// TIA Portal V17 export
// export: Created 2025-07-01T09:58:31.5693186Z, ExportSetting WithDefaults, DisplayName Totally Integrated Automation Portal, DisplayVersion V17 Update 8, DisplayName TIA Portal Openness, DisplayVersion V17 Update 8, DisplayName TIA Portal Version Control Interface, DisplayVersion V17, DisplayName SINAMICS Startdrive Advanced, DisplayVersion V17 SP2, DisplayName SINAMICS Startdrive G110M, G120, G120C, G120D, G120P, G115D, DisplayVersion V17 SP2, DisplayName SINAMICS Startdrive G130, G150, S120, S150, SINAMICS MV, S210, DisplayVersion V17 SP2, DisplayName STEP 7 Professional, DisplayVersion V17 Update 8, DisplayName SINUMERIK ONE STEP 7 Toolbox, DisplayVersion V17 Update 12, DisplayName SINUMERIK ONE PLC Basic Program Plus, DisplayVersion V17 Update 12, DisplayName SINUMERIK 840D sl STEP 7 Toolbox, DisplayVersion V17 Update 12, DisplayName STEP 7 Safety, DisplayVersion V17 Update 6, DisplayName WinCC Advanced, DisplayVersion V17 Update 8
FUNCTION "FC15500_BDE" : Void   // FC15500, LAD
{ S7_Optimized_Access := 'TRUE' }
VERSION : 0.1
// stored: AutoNumber false, IsIECCheckEnabled false, SetENOAutomatically false, UDAEnableTagReadback false
BEGIN

REGION Network 1: FEED PART STATUS
   // PART_A/PART_B/PART_C/PART_D/PART_E
   // If the bit for the status of a feed part is to 0, the corresponding message text+ is available
   // is displayed in the image.
   // If the bit for the status of a feed part is set to 1, the corresponding message text + not available is displayed on the screen.
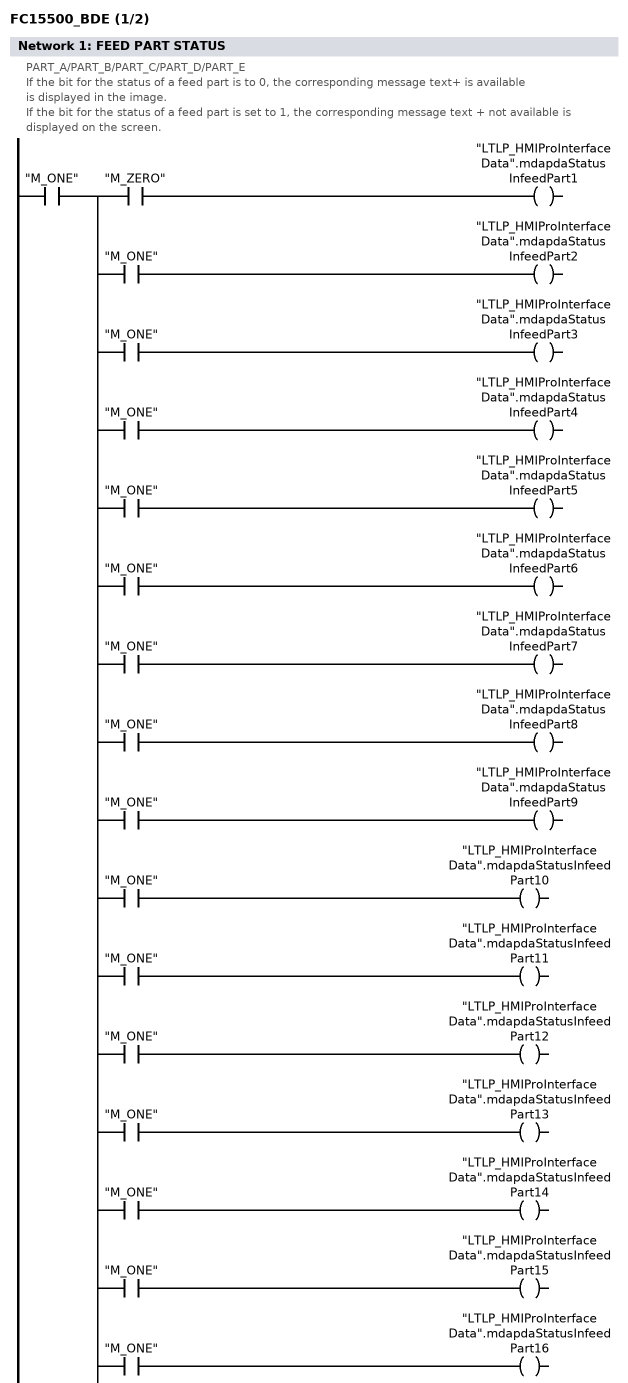
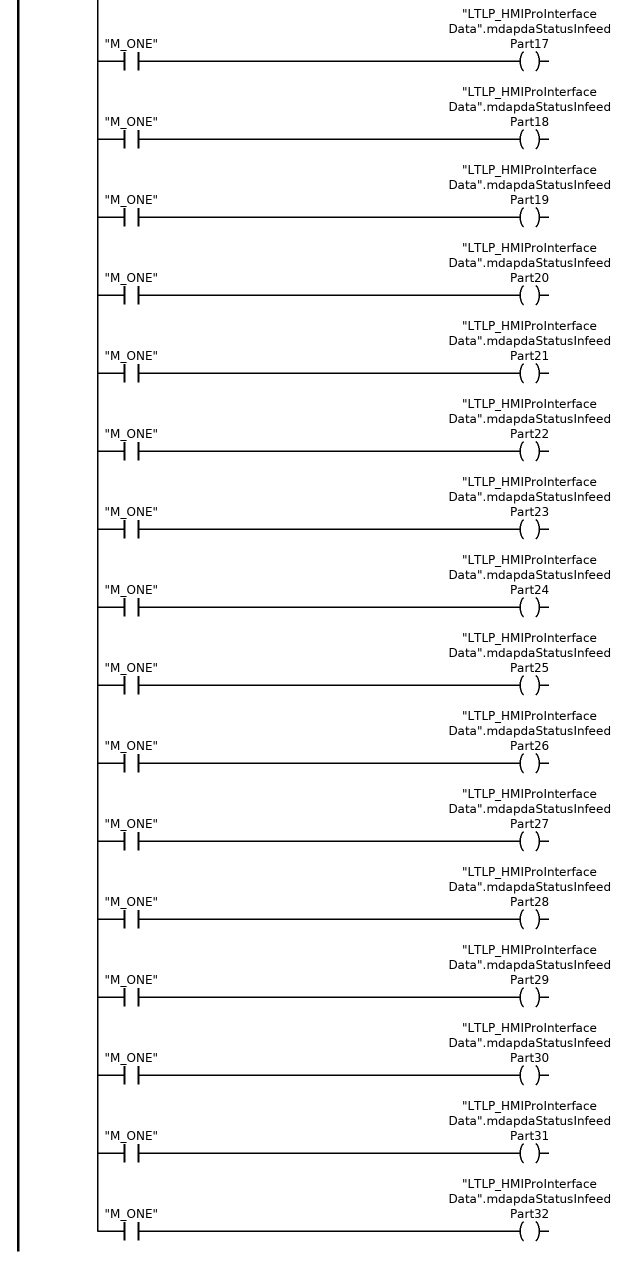
   RUNG wire#powerrail
      Contact( "M_ONE" )
      wire#w1
      Contact( "M_ZERO" )
      Coil( "LTLP_HMIProInterfaceData".mdapdaStatusInfeedPart1 )
   END_RUNG
   RUNG wire#w1
      Contact( "M_ONE" )
      Coil( "LTLP_HMIProInterfaceData".mdapdaStatusInfeedPart2 )
   END_RUNG
   RUNG wire#w1
      Contact( "M_ONE" )
      Coil( "LTLP_HMIProInterfaceData".mdapdaStatusInfeedPart3 )
   END_RUNG
   RUNG wire#w1
      Contact( "M_ONE" )
      Coil( "LTLP_HMIProInterfaceData".mdapdaStatusInfeedPart4 )
   END_RUNG
   RUNG wire#w1
      Contact( "M_ONE" )
      Coil( "LTLP_HMIProInterfaceData".mdapdaStatusInfeedPart5 )
   END_RUNG
   RUNG wire#w1
      Contact( "M_ONE" )
      Coil( "LTLP_HMIProInterfaceData".mdapdaStatusInfeedPart6 )
   END_RUNG
   RUNG wire#w1
      Contact( "M_ONE" )
      Coil( "LTLP_HMIProInterfaceData".mdapdaStatusInfeedPart7 )
   END_RUNG
   RUNG wire#w1
      Contact( "M_ONE" )
      Coil( "LTLP_HMIProInterfaceData".mdapdaStatusInfeedPart8 )
   END_RUNG
   RUNG wire#w1
      Contact( "M_ONE" )
      Coil( "LTLP_HMIProInterfaceData".mdapdaStatusInfeedPart9 )
   END_RUNG
   RUNG wire#w1
      Contact( "M_ONE" )
      Coil( "LTLP_HMIProInterfaceData".mdapdaStatusInfeedPart10 )
   END_RUNG
   RUNG wire#w1
      Contact( "M_ONE" )
      Coil( "LTLP_HMIProInterfaceData".mdapdaStatusInfeedPart11 )
   END_RUNG
   RUNG wire#w1
      Contact( "M_ONE" )
      Coil( "LTLP_HMIProInterfaceData".mdapdaStatusInfeedPart12 )
   END_RUNG
   RUNG wire#w1
      Contact( "M_ONE" )
      Coil( "LTLP_HMIProInterfaceData".mdapdaStatusInfeedPart13 )
   END_RUNG
   RUNG wire#w1
      Contact( "M_ONE" )
      Coil( "LTLP_HMIProInterfaceData".mdapdaStatusInfeedPart14 )
   END_RUNG
   RUNG wire#w1
      Contact( "M_ONE" )
      Coil( "LTLP_HMIProInterfaceData".mdapdaStatusInfeedPart15 )
   END_RUNG
   RUNG wire#w1
      Contact( "M_ONE" )
      Coil( "LTLP_HMIProInterfaceData".mdapdaStatusInfeedPart16 )
   END_RUNG
   RUNG wire#w1
      Contact( "M_ONE" )
      Coil( "LTLP_HMIProInterfaceData".mdapdaStatusInfeedPart17 )
   END_RUNG
   RUNG wire#w1
      Contact( "M_ONE" )
      Coil( "LTLP_HMIProInterfaceData".mdapdaStatusInfeedPart18 )
   END_RUNG
   RUNG wire#w1
      Contact( "M_ONE" )
      Coil( "LTLP_HMIProInterfaceData".mdapdaStatusInfeedPart19 )
   END_RUNG
   RUNG wire#w1
      Contact( "M_ONE" )
      Coil( "LTLP_HMIProInterfaceData".mdapdaStatusInfeedPart20 )
   END_RUNG
   RUNG wire#w1
      Contact( "M_ONE" )
      Coil( "LTLP_HMIProInterfaceData".mdapdaStatusInfeedPart21 )
   END_RUNG
   RUNG wire#w1
      Contact( "M_ONE" )
      Coil( "LTLP_HMIProInterfaceData".mdapdaStatusInfeedPart22 )
   END_RUNG
   RUNG wire#w1
      Contact( "M_ONE" )
      Coil( "LTLP_HMIProInterfaceData".mdapdaStatusInfeedPart23 )
   END_RUNG
   RUNG wire#w1
      Contact( "M_ONE" )
      Coil( "LTLP_HMIProInterfaceData".mdapdaStatusInfeedPart24 )
   END_RUNG
   RUNG wire#w1
      Contact( "M_ONE" )
      Coil( "LTLP_HMIProInterfaceData".mdapdaStatusInfeedPart25 )
   END_RUNG
   RUNG wire#w1
      Contact( "M_ONE" )
      Coil( "LTLP_HMIProInterfaceData".mdapdaStatusInfeedPart26 )
   END_RUNG
   RUNG wire#w1
      Contact( "M_ONE" )
      Coil( "LTLP_HMIProInterfaceData".mdapdaStatusInfeedPart27 )
   END_RUNG
   RUNG wire#w1
      Contact( "M_ONE" )
      Coil( "LTLP_HMIProInterfaceData".mdapdaStatusInfeedPart28 )
   END_RUNG
   RUNG wire#w1
      Contact( "M_ONE" )
      Coil( "LTLP_HMIProInterfaceData".mdapdaStatusInfeedPart29 )
   END_RUNG
   RUNG wire#w1
      Contact( "M_ONE" )
      Coil( "LTLP_HMIProInterfaceData".mdapdaStatusInfeedPart30 )
   END_RUNG
   RUNG wire#w1
      Contact( "M_ONE" )
      Coil( "LTLP_HMIProInterfaceData".mdapdaStatusInfeedPart31 )
   END_RUNG
   RUNG wire#w1
      Contact( "M_ONE" )
      Coil( "LTLP_HMIProInterfaceData".mdapdaStatusInfeedPart32 )
   END_RUNG
   // the same network as SCL:
   "LTLP_HMIProInterfaceData".mdapdaStatusInfeedPart1 := "M_ONE" AND "M_ZERO";
   "LTLP_HMIProInterfaceData".mdapdaStatusInfeedPart2 := "M_ONE" AND "M_ONE";
   "LTLP_HMIProInterfaceData".mdapdaStatusInfeedPart3 := "M_ONE" AND "M_ONE";
   "LTLP_HMIProInterfaceData".mdapdaStatusInfeedPart4 := "M_ONE" AND "M_ONE";
   "LTLP_HMIProInterfaceData".mdapdaStatusInfeedPart5 := "M_ONE" AND "M_ONE";
   "LTLP_HMIProInterfaceData".mdapdaStatusInfeedPart6 := "M_ONE" AND "M_ONE";
   "LTLP_HMIProInterfaceData".mdapdaStatusInfeedPart7 := "M_ONE" AND "M_ONE";
   "LTLP_HMIProInterfaceData".mdapdaStatusInfeedPart8 := "M_ONE" AND "M_ONE";
   "LTLP_HMIProInterfaceData".mdapdaStatusInfeedPart9 := "M_ONE" AND "M_ONE";
   "LTLP_HMIProInterfaceData".mdapdaStatusInfeedPart10 := "M_ONE" AND "M_ONE";
   "LTLP_HMIProInterfaceData".mdapdaStatusInfeedPart11 := "M_ONE" AND "M_ONE";
   "LTLP_HMIProInterfaceData".mdapdaStatusInfeedPart12 := "M_ONE" AND "M_ONE";
   "LTLP_HMIProInterfaceData".mdapdaStatusInfeedPart13 := "M_ONE" AND "M_ONE";
   "LTLP_HMIProInterfaceData".mdapdaStatusInfeedPart14 := "M_ONE" AND "M_ONE";
   "LTLP_HMIProInterfaceData".mdapdaStatusInfeedPart15 := "M_ONE" AND "M_ONE";
   "LTLP_HMIProInterfaceData".mdapdaStatusInfeedPart16 := "M_ONE" AND "M_ONE";
   "LTLP_HMIProInterfaceData".mdapdaStatusInfeedPart17 := "M_ONE" AND "M_ONE";
   "LTLP_HMIProInterfaceData".mdapdaStatusInfeedPart18 := "M_ONE" AND "M_ONE";
   "LTLP_HMIProInterfaceData".mdapdaStatusInfeedPart19 := "M_ONE" AND "M_ONE";
   "LTLP_HMIProInterfaceData".mdapdaStatusInfeedPart20 := "M_ONE" AND "M_ONE";
   "LTLP_HMIProInterfaceData".mdapdaStatusInfeedPart21 := "M_ONE" AND "M_ONE";
   "LTLP_HMIProInterfaceData".mdapdaStatusInfeedPart22 := "M_ONE" AND "M_ONE";
   "LTLP_HMIProInterfaceData".mdapdaStatusInfeedPart23 := "M_ONE" AND "M_ONE";
   "LTLP_HMIProInterfaceData".mdapdaStatusInfeedPart24 := "M_ONE" AND "M_ONE";
   "LTLP_HMIProInterfaceData".mdapdaStatusInfeedPart25 := "M_ONE" AND "M_ONE";
   "LTLP_HMIProInterfaceData".mdapdaStatusInfeedPart26 := "M_ONE" AND "M_ONE";
   "LTLP_HMIProInterfaceData".mdapdaStatusInfeedPart27 := "M_ONE" AND "M_ONE";
   "LTLP_HMIProInterfaceData".mdapdaStatusInfeedPart28 := "M_ONE" AND "M_ONE";
   "LTLP_HMIProInterfaceData".mdapdaStatusInfeedPart29 := "M_ONE" AND "M_ONE";
   "LTLP_HMIProInterfaceData".mdapdaStatusInfeedPart30 := "M_ONE" AND "M_ONE";
   "LTLP_HMIProInterfaceData".mdapdaStatusInfeedPart31 := "M_ONE" AND "M_ONE";
   "LTLP_HMIProInterfaceData".mdapdaStatusInfeedPart32 := "M_ONE" AND "M_ONE";
END_REGION

REGION Network 2: STATUS - SWITCHED ON/OFF
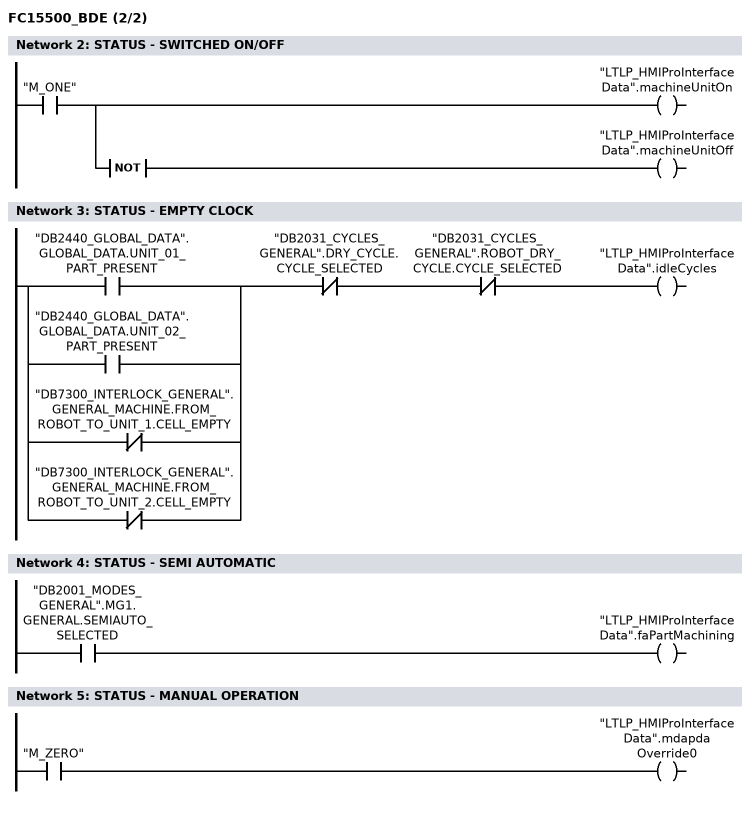
   RUNG wire#powerrail
      Contact( "M_ONE" )
      wire#w1
      Coil( "LTLP_HMIProInterfaceData".machineUnitOn )
   END_RUNG
   RUNG wire#w1
      Not()
      Coil( "LTLP_HMIProInterfaceData".machineUnitOff )
   END_RUNG
   // the same network as SCL:
   "LTLP_HMIProInterfaceData".machineUnitOn := "M_ONE";
   "LTLP_HMIProInterfaceData".machineUnitOff := NOT "M_ONE";
END_REGION

REGION Network 3: STATUS - EMPTY CLOCK
   RUNG wire#powerrail
      Contact( "DB2440_GLOBAL_DATA".GLOBAL_DATA.UNIT_01_PART_PRESENT )
      wire#w1
      I_Contact( "DB2031_CYCLES_GENERAL".DRY_CYCLE.CYCLE_SELECTED )
      I_Contact( "DB2031_CYCLES_GENERAL".ROBOT_DRY_CYCLE.CYCLE_SELECTED )
      Coil( "LTLP_HMIProInterfaceData".idleCycles )
   END_RUNG
   RUNG wire#powerrail
      Contact( "DB2440_GLOBAL_DATA".GLOBAL_DATA.UNIT_02_PART_PRESENT )
   END_RUNG wire#w1
   RUNG wire#powerrail
      I_Contact( "DB7300_INTERLOCK_GENERAL".GENERAL_MACHINE.FROM_ROBOT_TO_UNIT_1.CELL_EMPTY )
   END_RUNG wire#w1
   RUNG wire#powerrail
      I_Contact( "DB7300_INTERLOCK_GENERAL".GENERAL_MACHINE.FROM_ROBOT_TO_UNIT_2.CELL_EMPTY )
   END_RUNG wire#w1
   // the same network as SCL:
   "LTLP_HMIProInterfaceData".idleCycles := ("DB2440_GLOBAL_DATA".GLOBAL_DATA.UNIT_01_PART_PRESENT OR "DB2440_GLOBAL_DATA".GLOBAL_DATA.UNIT_02_PART_PRESENT OR NOT "DB7300_INTERLOCK_GENERAL".GENERAL_MACHINE.FROM_ROBOT_TO_UNIT_1.CELL_EMPTY OR NOT "DB7300_INTERLOCK_GENERAL".GENERAL_MACHINE.FROM_ROBOT_TO_UNIT_2.CELL_EMPTY) AND NOT "DB2031_CYCLES_GENERAL".DRY_CYCLE.CYCLE_SELECTED AND NOT "DB2031_CYCLES_GENERAL".ROBOT_DRY_CYCLE.CYCLE_SELECTED;
END_REGION

REGION Network 4: STATUS - SEMI AUTOMATIC
   RUNG wire#powerrail
      Contact( "DB2001_MODES_GENERAL".MG1.GENERAL.SEMIAUTO_SELECTED )
      Coil( "LTLP_HMIProInterfaceData".faPartMachining )
   END_RUNG
   // the same network as SCL:
   "LTLP_HMIProInterfaceData".faPartMachining := "DB2001_MODES_GENERAL".MG1.GENERAL.SEMIAUTO_SELECTED;
END_REGION

REGION Network 5: STATUS - MANUAL OPERATION
   RUNG wire#powerrail
      Contact( "M_ZERO" )
      Coil( "LTLP_HMIProInterfaceData".mdapdaOverride0 )
   END_RUNG
   // the same network as SCL:
   "LTLP_HMIProInterfaceData".mdapdaOverride0 := "M_ZERO";
END_REGION
END_FUNCTION
